VAR_GLOBAL CONSTANT
	/// ctrl commands definitions
	/// specific commands >200 - every command has to be a even number
	cBCC_CMD_READ: INT 	:= 202;
	/// ctrl specific states definitions
	cBCC_STA_READBusy	: INT := 201;
	cBCC_STA_READ		: INT := cBCC_CMD_READ;
END_VAR

(* stored: Version 1.1.0.1, ProductVersion 3.1.0.26
   GVL BCC_CmdState: Id {c7ec8444-7fde-48d7-a68b-5e5b7dcde440} *)
